INTERFACE I_Read_Only_Line_Builder_Adapter EXTENDS T_Query_Interface

END_INTERFACE

(* stored: Version 1.1.0.1, ProductVersion 3.1.4024.4
   Itf I_Read_Only_Line_Builder_Adapter: Id {691d2814-da6a-4beb-b2ce-accd421bc0f6} *)
